// TIA Portal V19 export
TYPE "LEXCHANGETRAY_typeScanner_controlInterface"
// stored: Access Published
   STRUCT
      cmd : "LEXCHANGETRAY_typeScanner_cmd";
      par : "LEXCHANGETRAY_typeScanner_par";
      monitor : "LEXCHANGETRAY_typeScanner_monitor";
      sim : "LEXCHANGETRAY_typeScanner_sim";
   END_STRUCT;
END_TYPE
